							str_response:=concat(byte_to_hexstr(a_response[0],2,TRUE),byte_to_hexstr(a_response[1],2,TRUE));
							str_response:=concat(str_response,byte_to_hexstr(a_response[2],2,TRUE));
							str_response:=concat(str_response,byte_to_hexstr(a_response[3],2,TRUE));
							str_response:=concat(str_response,byte_to_hexstr(a_response[4],2,TRUE));
							str_response:=concat(str_response,byte_to_hexstr(a_response[5],2,TRUE));
							str_response:=concat(str_response,byte_to_hexstr(a_response[6],2,TRUE));
							str_response:=concat(str_response,byte_to_hexstr(a_response[7],2,TRUE));
							str_response:=concat(str_response,byte_to_hexstr(a_response[8],2,TRUE));
							str_response:=concat(str_response,byte_to_hexstr(a_response[9],2,TRUE));
							str_response:=concat(str_response,byte_to_hexstr(a_response[10],2,TRUE));
							str_response:=concat(str_response,byte_to_hexstr(a_response[11],2,TRUE));
							str_response:=concat(str_response,byte_to_hexstr(a_response[12],2,TRUE));
							str_response:=concat(str_response,byte_to_hexstr(a_response[13],2,TRUE));
							str_response:=concat(str_response,byte_to_hexstr(a_response[14],2,TRUE));
							str_response:=concat(str_response,byte_to_hexstr(a_response[15],2,TRUE));
							str_response:=concat(str_response,byte_to_hexstr(a_response[16],2,TRUE));
							str_response:=concat(str_response,byte_to_hexstr(a_response[17],2,TRUE));
							str_response:=concat(str_response,byte_to_hexstr(a_response[18],2,TRUE));
							str_response:=concat(str_response,byte_to_hexstr(a_response[19],2,TRUE));
							str_response:=concat(str_response,byte_to_hexstr(a_response[20],2,TRUE));
							str_response:=concat(str_response,byte_to_hexstr(a_response[21],2,TRUE));
							str_response:=concat(str_response,byte_to_hexstr(a_response[22],2,TRUE));
							str_response:=concat(str_response,byte_to_hexstr(a_response[23],2,TRUE));
							str_response:=concat(str_response,byte_to_hexstr(a_response[24],2,TRUE));
							str_response:=concat(str_response,byte_to_hexstr(a_response[25],2,TRUE));
							str_response:=concat(str_response,byte_to_hexstr(a_response[26],2,TRUE));
							str_response:=concat(str_response,byte_to_hexstr(a_response[27],2,TRUE));
							str_response:=concat(str_response,byte_to_hexstr(a_response[28],2,TRUE));
							str_response:=concat(str_response,byte_to_hexstr(a_response[29],2,TRUE));
							str_response:=concat(str_response,byte_to_hexstr(a_response[30],2,TRUE));
							str_response:=concat(str_response,byte_to_hexstr(a_response[31],2,TRUE));
							
						// "Digest username=\"admin\", realm=\"shellypro4pm-083af27cfbac\", nonce=\"63768368\", uri=\"/rpc/Switch.GetStatus?id=0\", algorithm=\"SHA-256\", qop=auth, nc=00000001, cnonce=\"oKOklSrS\", response=\"d1d59d1e015dee0a3acfc97b20a0fa0ff851b03d79ca00df59ce018a63041468\""
						
						str_authorization:=concat('Digest username="admin", realm="',sRealm);
						str_authorization:=concat(str_authorization,'", nonce="');
						str_authorization:=concat(str_authorization,snonce);
						str_authorization:=concat(str_authorization,'", algorithm="SHA-256", uri="/rpc/Switch.Set?id=0&on=FALSE", qop=auth, nc=00000001, cnonce="');
						str_authorization:=concat(str_authorization,scnonce);
						str_authorization:=concat(str_authorization,'", response="');
						str_authorization:=concat(str_authorization,str_response);
						str_authorization:=concat(str_authorization,'"');
						
						fbHeader2.AddField('Authorization', str_authorization, FALSE);
						IF fbRequest3.SendRequest(sUri:= '/rpc/Switch.Set?id=0&on=FALSE', fbClient:= fbClient, eRequestType:= ETcIotHttpRequestType.HTTP_Get, 0, 0, fbHeader2) THEN
							nState:= 5;
							bBusy:= TRUE;
							bError:= FALSE;
						END_IF
				END_IF
			END_IF
		END_IF
	5:	
		IF bSetOnP1 AND NOT bStateP1 THEN 
			IF
				fbRequest3.SendRequest(sUri:='/rpc/Switch.Set?id=0&on=true', fbClient:=fbClient, eRequestType:=ETcIotHttpRequestType.HTTP_Get, 0, 0, fbHeader2) THEN				
				bSetOnP1 := FALSE;
				int_CountOnWrite := int_CountOnWrite +1;
				nState:= 6;
				bBusy:= TRUE;
				bError:= FALSE;
			END_IF					
		ELSIF bSetOffP1 AND bStateP1 THEN 
			IF	
				fbRequest3.SendRequest(sUri:='/rpc/Switch.Set?id=0&on=false', fbClient:=fbClient, eRequestType:=ETcIotHttpRequestType.HTTP_Get, 0, 0, fbHeader2) THEN				
				bSetOffP1 := FALSE;
				int_CountOffWrite := int_CountOffWrite +1;
				nState:= 6;
				bBusy:= TRUE;
				bError:= FALSE;
			END_IF	
		ELSE
			nState:= 6;
		END_IF
	6:
		bBusy:= FALSE;
		nState:= 0;

	
END_CASE

END_FUNCTION_BLOCK

// ---- POUs/prgRWEffIO.TcPOU
PROGRAM prgRWEffIO
VAR
	fbRW1		: FB_ReadWrite_V2;
END_VAR


fbRW1(
	eUploadType:= 3, // Change + 5 min Intervall 
	bBusy=> , 
	bError=> , 
	udiErrorCodeOut=> , 
	eErrorReadWrite_Out=> );

END_PROGRAM
